(* PLC project Generated.project, CODESYS CODESYS V3.5 SP19 Patch 1 *)
(* stored: creationDateTime 2026-09-01T00:57:57.826716, modificationDateTime 2026-09-01T00:57:57.826716 *)

(* ═══════════════════════════════════════════════════════════════ 🎮 ST_CycleExtractionCmd — Sélections IHM cycle extraction ═══════════════════════════════════════════════════════════════ *)
TYPE ST_CycleExtractionCmd : STRUCT
  TglEnableExtractionSequence : BOOL := FALSE;  (* Assistance extraction active *)
END_STRUCT;
END_TYPE
